Fanuc KAREL source: kt00376.KL

-- PROVISIONAL review KL for V940-1; original PC SHA256 ce0334e5c39df4ac1292a72d877854a253535cd293927e9b7fa414a22aa03031
-- Incomplete behavior may be omitted. Consult companion uncertainty JSON. Do not deploy.
PROGRAM KT00376
%NOLOCKGROUP
VAR
  R2 : REAL
  OUT : BOOLEAN
-- UNRESOLVED_DECL Y1 type=002018
BEGIN
  -- V9_ZERO_TABLE_METADATA_HINT layout=0001; no indexed target words; source/name/runtime held
  -- UNRESOLVED_PC offsets 5-19; opcodes 2E,22,9D,33,B2
  -- UNRESOLVED_PC offsets 24-35; opcodes 2E,23
  -- UNRESOLVED_PC offsets 40-65; opcodes 22,9D,33,B1,21,29,64,29,70,23
  -- UNRESOLVED_PC offsets 70-74; opcodes 7F
END KT00376
